PROGRAM PRG_PLAS_04_CompleteOuterCtrl
VAR
	rsShiftOCVDataControl			: RS;
	fbMoveOuterStatusArray			: FB_PACK_MoveOuterStatusArray;
	fbAddNewOCVTriggerID			: FB_PLAS_AddNewTriggerID;
	fbCompleteOCV  					: FB_T01_CompleteOCV;

	tofWarningForStacker				: TOF;
	ctuArmAtBackwardPosition		: FB_CTU32;

	nIndexTreshold					: UDINT := 5;
	nTransferIndex						: UDINT ;

	ctuConsecutiveIntermediateNoRead		: CTU;
	ctuConsecutiveOCVMissing				: CTU;

	fbDebugCNT						: FB_DEBUG_CounterArray;
	aCNTDebug						: ARRAY [1..10] OF UDINT;
	bResetCNT							: BOOL;
END_VAR

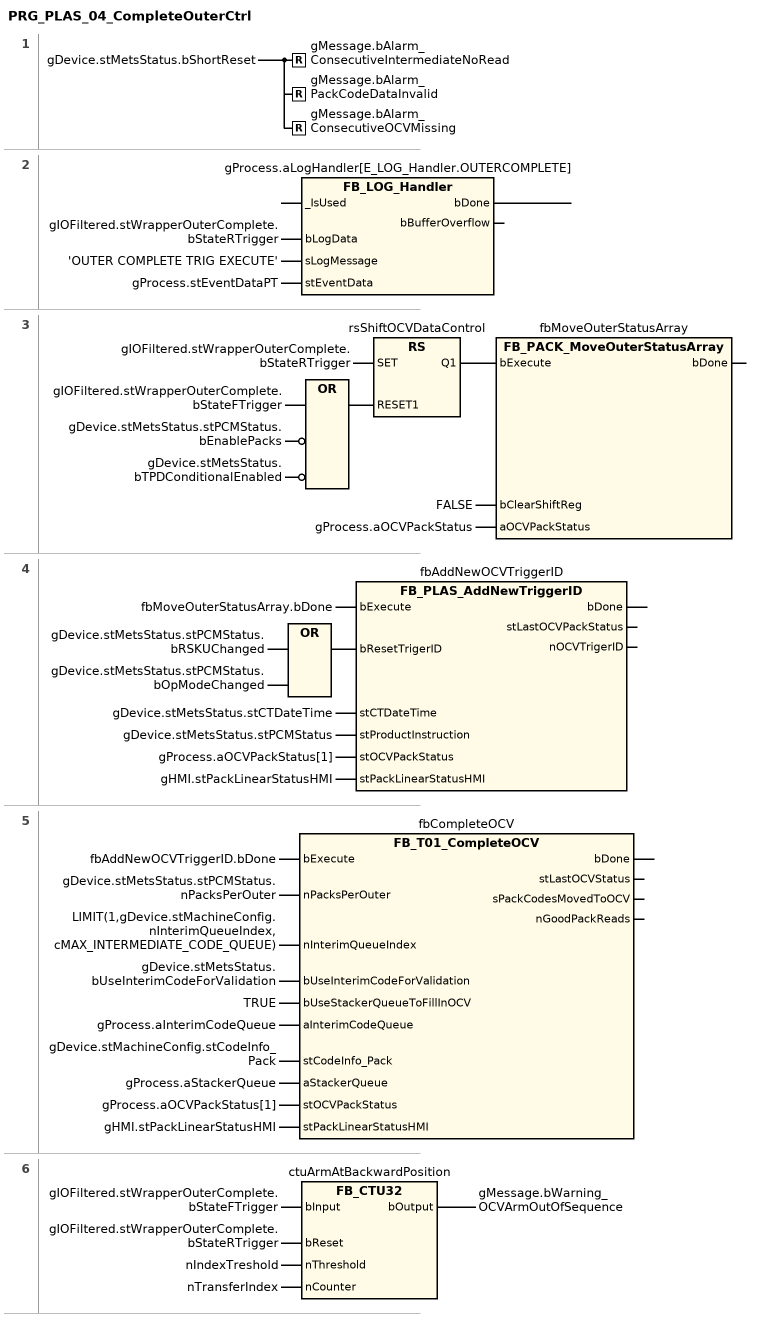
// NETWORK 1
gMessage.bAlarm_ConsecutiveIntermediateNoRead R= gDevice.stMetsStatus.bShortReset;
gMessage.bAlarm_PackCodeDataInvalid R= gDevice.stMetsStatus.bShortReset;
gMessage.bAlarm_ConsecutiveOCVMissing R= gDevice.stMetsStatus.bShortReset;

// NETWORK 2
gProcess.aLogHandler[E_LOG_Handler.OUTERCOMPLETE](
    bLogData := gIOFiltered.stWrapperOuterComplete.bStateRTrigger,
    sLogMessage := 'OUTER COMPLETE TRIG EXECUTE',
    stEventData := gProcess.stEventDataPT); // FB_LOG_Handler

// NETWORK 3
rsShiftOCVDataControl(SET := gIOFiltered.stWrapperOuterComplete.bStateRTrigger, RESET1 := gIOFiltered.stWrapperOuterComplete.bStateFTrigger OR NOT gDevice.stMetsStatus.stPCMStatus.bEnablePacks OR NOT gDevice.stMetsStatus.bTPDConditionalEnabled); // RS
fbMoveOuterStatusArray(
    bExecute := rsShiftOCVDataControl.Q1,
    bClearShiftReg := FALSE,
    aOCVPackStatus := gProcess.aOCVPackStatus); // FB_PACK_MoveOuterStatusArray

// NETWORK 4
fbAddNewOCVTriggerID(
    bExecute := fbMoveOuterStatusArray.bDone,
    bResetTrigerID := gDevice.stMetsStatus.stPCMStatus.bRSKUChanged OR gDevice.stMetsStatus.stPCMStatus.bOpModeChanged,
    stCTDateTime := gDevice.stMetsStatus.stCTDateTime,
    stProductInstruction := gDevice.stMetsStatus.stPCMStatus,
    stOCVPackStatus := gProcess.aOCVPackStatus[1],
    stPackLinearStatusHMI := gHMI.stPackLinearStatusHMI); // FB_PLAS_AddNewTriggerID

// NETWORK 5
fbCompleteOCV(
    bExecute := fbAddNewOCVTriggerID.bDone,
    nPacksPerOuter := gDevice.stMetsStatus.stPCMStatus.nPacksPerOuter,
    nInterimQueueIndex := LIMIT(1,gDevice.stMachineConfig.nInterimQueueIndex, cMAX_INTERMEDIATE_CODE_QUEUE),
    bUseInterimCodeForValidation := gDevice.stMetsStatus.bUseInterimCodeForValidation,
    bUseStackerQueueToFillInOCV := TRUE,
    aInterimCodeQueue := gProcess.aInterimCodeQueue,
    stCodeInfo_Pack := gDevice.stMachineConfig.stCodeInfo_Pack,
    aStackerQueue := gProcess.aStackerQueue,
    stOCVPackStatus := gProcess.aOCVPackStatus[1],
    stPackLinearStatusHMI := gHMI.stPackLinearStatusHMI); // FB_T01_CompleteOCV

// NETWORK 6
ctuArmAtBackwardPosition(
    bInput := gIOFiltered.stWrapperOuterComplete.bStateFTrigger,
    bReset := gIOFiltered.stWrapperOuterComplete.bStateRTrigger,
    nThreshold := nIndexTreshold,
    nCounter := nTransferIndex); // FB_CTU32
gMessage.bWarning_OCVArmOutOfSequence := ctuArmAtBackwardPosition.bOutput;

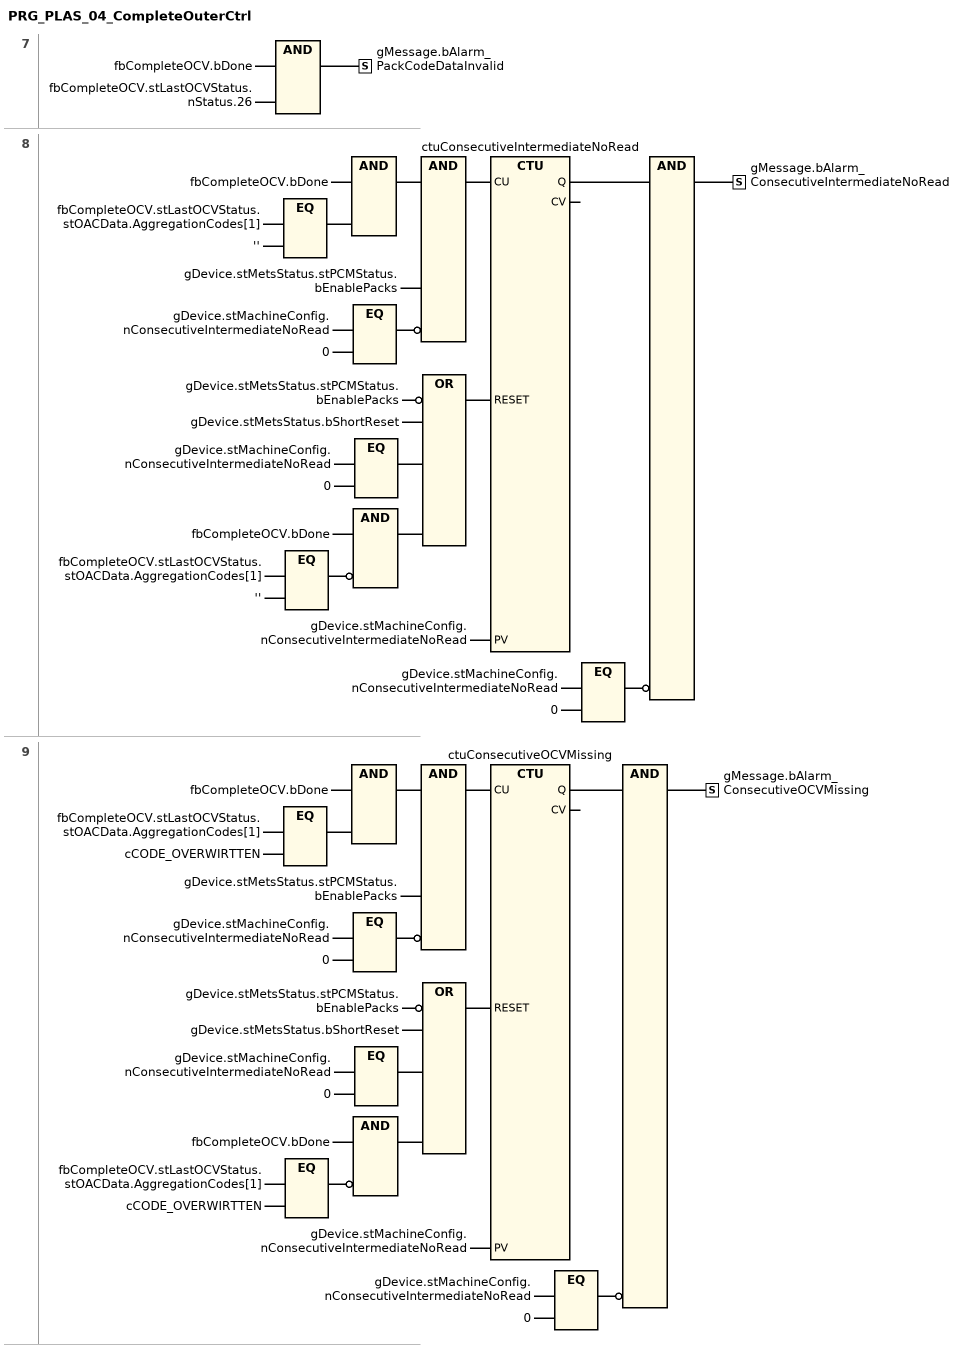
// NETWORK 7
gMessage.bAlarm_PackCodeDataInvalid S= fbCompleteOCV.bDone AND fbCompleteOCV.stLastOCVStatus.nStatus.26;

// NETWORK 8
ctuConsecutiveIntermediateNoRead(
    CU := (fbCompleteOCV.bDone AND fbCompleteOCV.stLastOCVStatus.stOACData.AggregationCodes[1] = '') AND gDevice.stMetsStatus.stPCMStatus.bEnablePacks AND NOT (gDevice.stMachineConfig.nConsecutiveIntermediateNoRead = 0),
    RESET := NOT gDevice.stMetsStatus.stPCMStatus.bEnablePacks OR gDevice.stMetsStatus.bShortReset OR gDevice.stMachineConfig.nConsecutiveIntermediateNoRead = 0 OR fbCompleteOCV.bDone AND NOT (fbCompleteOCV.stLastOCVStatus.stOACData.AggregationCodes[1] = ''),
    PV := gDevice.stMachineConfig.nConsecutiveIntermediateNoRead); // CTU
gMessage.bAlarm_ConsecutiveIntermediateNoRead S= ctuConsecutiveIntermediateNoRead.Q AND NOT (gDevice.stMachineConfig.nConsecutiveIntermediateNoRead = 0);

// NETWORK 9
ctuConsecutiveOCVMissing(
    CU := (fbCompleteOCV.bDone AND fbCompleteOCV.stLastOCVStatus.stOACData.AggregationCodes[1] = cCODE_OVERWIRTTEN) AND gDevice.stMetsStatus.stPCMStatus.bEnablePacks AND NOT (gDevice.stMachineConfig.nConsecutiveIntermediateNoRead = 0),
    RESET := NOT gDevice.stMetsStatus.stPCMStatus.bEnablePacks OR gDevice.stMetsStatus.bShortReset OR gDevice.stMachineConfig.nConsecutiveIntermediateNoRead = 0 OR fbCompleteOCV.bDone AND NOT (fbCompleteOCV.stLastOCVStatus.stOACData.AggregationCodes[1] = cCODE_OVERWIRTTEN),
    PV := gDevice.stMachineConfig.nConsecutiveIntermediateNoRead); // CTU
gMessage.bAlarm_ConsecutiveOCVMissing S= ctuConsecutiveOCVMissing.Q AND NOT (gDevice.stMachineConfig.nConsecutiveIntermediateNoRead = 0);

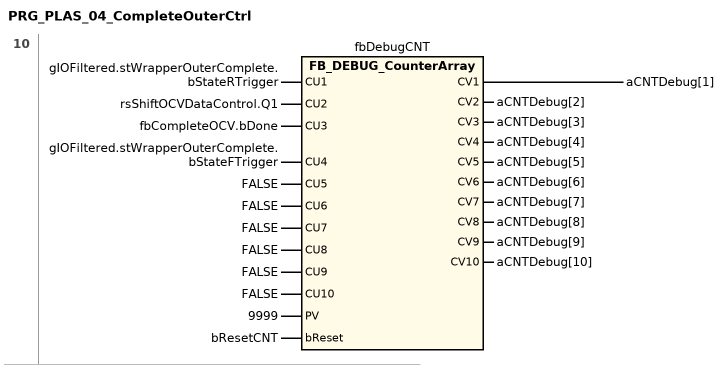
// NETWORK 10
fbDebugCNT(
    CU1 := gIOFiltered.stWrapperOuterComplete.bStateRTrigger,
    CU2 := rsShiftOCVDataControl.Q1,
    CU3 := fbCompleteOCV.bDone,
    CU4 := gIOFiltered.stWrapperOuterComplete.bStateFTrigger,
    CU5 := FALSE,
    CU6 := FALSE,
    CU7 := FALSE,
    CU8 := FALSE,
    CU9 := FALSE,
    CU10 := FALSE,
    PV := 9999,
    bReset := bResetCNT,
    CV2 => aCNTDebug[2],
    CV3 => aCNTDebug[3],
    CV4 => aCNTDebug[4],
    CV5 => aCNTDebug[5],
    CV6 => aCNTDebug[6],
    CV7 => aCNTDebug[7],
    CV8 => aCNTDebug[8],
    CV9 => aCNTDebug[9],
    CV10 => aCNTDebug[10]); // FB_DEBUG_CounterArray
aCNTDebug[1] := fbDebugCNT.CV1;

END_PROGRAM

(* stored: Version 1.1.0.1
   POU PRG_PLAS_04_CompleteOuterCtrl: Id {f38a8eb6-2632-44ca-a01f-ecf644a3118d}, SpecialFunc None *)
